FUNCTION_BLOCK TRAFFICCONTROL1 (* Basic Function Block Type *)
  (* Standard: 61499-2 *)
  (* Version 0.3, 2009-09-15, JHC, Holobloc Inc, Changed transition priorities. *)
  (* Version 0.2, 2003-12-04, JHC, Rockwell Automation, Renamed for better indexing. *)
  (* Version 0.1, 2002-11-05, JHC, Rockwell Automation, Corrected missing ST element in Algorithm REQ. *)
  (* Version 0.0, 2000-05-30, JHC, Rockwell Automation *)
  (* Compiler header: package fb.rt.template; *)
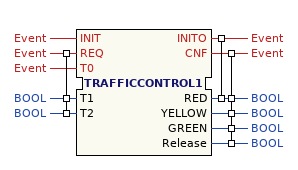
  EVENT_INPUT
    INIT; (* Initialization Request *)
    REQ WITH T1, T2; (* Normal Execution Request *)
    T0;
  END_EVENT
  EVENT_OUTPUT
    INITO WITH RED; (* Initialization Confirm *)
    CNF WITH RED, YELLOW, GREEN, Release; (* Execution Confirmation *)
  END_EVENT
  VAR_INPUT
    T1 : BOOL;
    T2 : BOOL;
  END_VAR
  VAR_OUTPUT
    RED : BOOL; (* Output event qualifier *)
    YELLOW : BOOL;
    GREEN : BOOL;
    Release : BOOL;
  END_VAR
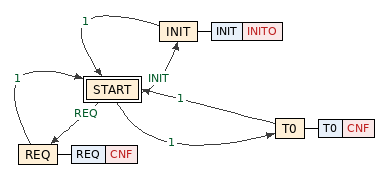
  EC_STATES
    START; (* Initial State *)
    INIT : INIT -> INITO; (* Initialization *)
    REQ : REQ -> CNF; (* Normal execution *)
    T0 : T0 -> CNF;
  END_STATES
  EC_TRANSITIONS
    INIT TO START := 1;
    START TO REQ := REQ;
    START TO INIT := INIT;
    REQ TO START := 1;
    START TO T0 := 1;
    T0 TO START := 1;
  END_TRANSITIONS
  ALGORITHM INIT IN ST: (* Initialization algorithm *)
GREEN:=FALSE;
YELLOW:=FALSE;
RED:=FALSE;
Release:=FALSE;
  END_ALGORITHM
  ALGORITHM REQ IN ST: (* Normally executed algorithm *)
IF T2 THEN
	YELLOW:=FALSE;
	RED:=TRUE;
  	Release:=TRUE;
ELSIF T1 THEN
	GREEN:=FALSE;
	YELLOW:=TRUE;
END_IF;
  END_ALGORITHM
  ALGORITHM T0 IN ST:
GREEN:=TRUE;
YELLOW:=FALSE;
RED:=FALSE;
Release:=FALSE;
  END_ALGORITHM
END_FUNCTION_BLOCK
